// TwinCAT 3 PLC project AdsGo_Det
// ProgramVersion: 3.1.4026.21
// libraries:
//   Tc2_Standard, * (Beckhoff Automation GmbH)
//   Tc2_System, * (Beckhoff Automation GmbH)
//   Tc3_Module, * (Beckhoff Automation GmbH)
// project tree:
//   Lib/ TestStruct.TcDUT, PackNone.TcDUT, PackTwo.TcDUT, PackFour.TcDUT, PackEight.TcDUT, StructTests.TcPOU, Deterministic.TcPOU
//   Programs/ Main.TcPOU
//   Tasks/ PlcTask.TcTTO
// real-time tasks:
//   TASK PlcTask: cycle T#10ms, priority 20, ADS port 354

CONFIGURATION AdsGo_Det
    RESOURCE PLC ON TwinCAT3
        TASK PlcTask(INTERVAL := T#10ms, PRIORITY := 20);
        PROGRAM Main WITH PlcTask : Main;
    END_RESOURCE
END_CONFIGURATION

// ---- Lib/TestStruct.TcDUT
TYPE TestStruct :
STRUCT
	seed       : UDINT;
	bool_var   : BOOL;
	sint_var   : SINT;
	usint_var  : USINT;
	byte_var   : BYTE;
	int_var    : INT;
	uint_var   : UINT;
	word_var   : WORD;
	dint_var   : DINT;
	udint_var  : UDINT;
	dword_var  : DWORD;
	lint_var   : LINT;
	ulint_var  : ULINT;
	lword_var  : LWORD;
	real_var   : REAL;
	lreal_var  : LREAL;
	time_var   : TIME;
	tod_var    : TOD;
	date_var   : DATE;
	dt_var     : DT;
	//ltime_var : LTIME;
	//ltod_var  : LTOD;
	//ldate_var : LDATE;
	//ldt_var   : LDT;
	string_var : STRING(255);
END_STRUCT
END_TYPE

// ---- Lib/PackNone.TcDUT
{attribute 'pack_mode' := '0'}
TYPE PackNone :
STRUCT
	b1  : BOOL;
	d1  : DWORD;
	b2  : BOOL;
	lw1 : LWORD;
END_STRUCT
END_TYPE

// ---- Lib/PackTwo.TcDUT
{attribute 'pack_mode' := '2'}
TYPE PackTwo :
STRUCT
	b1  : BOOL;
	d1  : DWORD;
	b2  : BOOL;
	lw1 : LWORD;
END_STRUCT
END_TYPE

// ---- Lib/PackFour.TcDUT
{attribute 'pack_mode' := '4'}
TYPE PackFour :
STRUCT
	b1  : BOOL;
	d1  : DWORD;
	b2  : BOOL;
	lw1 : LWORD;
END_STRUCT
END_TYPE

// ---- Lib/PackEight.TcDUT
{attribute 'pack_mode' := '8'}
TYPE PackEight :
STRUCT
	b1  : BOOL;
	d1  : DWORD;
	b2  : BOOL;
	lw1 : LWORD;
END_STRUCT
END_TYPE

// ---- Programs/Main.TcPOU
PROGRAM Main
VAR
	test : Deterministic;

	// Writable targets — PLC never modifies these, Go test owns them
	write_bool_var   : BOOL;
	write_sint_var   : SINT;
	write_usint_var  : USINT;
	write_byte_var   : BYTE;
	write_int_var    : INT;
	write_uint_var   : UINT;
	write_word_var   : WORD;
	write_dint_var   : DINT;
	write_udint_var  : UDINT;
	write_dword_var  : DWORD;
	write_lint_var   : LINT;
	write_ulint_var  : ULINT;
	write_lword_var  : LWORD;
	write_real_var   : REAL;
	write_lreal_var  : LREAL;
	write_time_var   : TIME;
	write_tod_var    : TOD;
	write_date_var   : DATE;
	write_dt_var     : DT;
	//write_ltime_var  : LTIME;
	//write_ltod_var   : LTOD;
	//write_ldate_var  : LDATE;
	//write_ldt_var    : LDT;
	write_string_var : STRING(255);
	write_struct_var : TestStruct;
	write_int_array  : ARRAY[0..9] OF INT;
	write_dint_array : ARRAY[0..9] OF DINT;
	write_2d_array   : ARRAY[0..2, 0..2] OF INT;

	// Struct packing test targets — one instance per pack_mode
	// struct_tests: PLC drives these from seed (Go read-only for phase 1)
	struct_tests : StructTests;
	// pack_*: Go-owned write targets (PLC never modifies, used in phase 2)
	pack_none  : PackNone;
	pack_two   : PackTwo;
	pack_four  : PackFour;
	pack_eight : PackEight;
END_VAR

test();
struct_tests();

END_PROGRAM

// ---- Lib/Deterministic.TcPOU
FUNCTION_BLOCK Deterministic
VAR
	// Control (writable by Go test)
	seed               : UDINT := 0;
	auto_mode          : BOOL := FALSE;
	auto_tick_interval : UDINT := 50;

	// Outputs
	bool_var   : BOOL;
	sint_var   : SINT;
	usint_var  : USINT;
	byte_var   : BYTE;
	int_var    : INT;
	uint_var   : UINT;
	word_var   : WORD;
	dint_var   : DINT;
	udint_var  : UDINT;
	dword_var  : DWORD;
	lint_var   : LINT;
	ulint_var  : ULINT;
	lword_var  : LWORD;
	real_var   : REAL;
	lreal_var  : LREAL;
	time_var   : TIME;
	tod_var    : TOD;
	date_var   : DATE;
	dt_var     : DT;
	//ltime_var  : LTIME;
	//ltod_var   : LTOD;
	//ldate_var  : LDATE;
	//ldt_var    : LDT;
	string_var : STRING(255);
	struct_var : TestStruct;
	int_array  : ARRAY[0..9] OF INT;
	dint_array : ARRAY[0..9] OF DINT;
	array_2d   : ARRAY[0..2, 0..2] OF INT;

	// Private
	_tick_counter : UDINT;
	_i            : UDINT;
	_j            : UDINT;
END_VAR

// -----------------------------------------------------------------------
// Auto-increment mode: advance seed every auto_tick_interval cycles
// -----------------------------------------------------------------------
IF auto_mode THEN
	IF _tick_counter >= auto_tick_interval THEN
		seed          := seed + 1;
		_tick_counter := 0;
	ELSE
		_tick_counter := _tick_counter + 1;
	END_IF
END_IF

// -----------------------------------------------------------------------
// Update variables — all fields are deterministic functions of seed
// -----------------------------------------------------------------------
bool_var  := (seed MOD 2 = 0);
sint_var  := UDINT_TO_SINT(seed);
usint_var := UDINT_TO_USINT(seed);
byte_var  := UDINT_TO_BYTE(seed);
int_var   := UDINT_TO_INT(seed);
uint_var  := UDINT_TO_UINT(seed);
word_var  := UDINT_TO_WORD(seed);
dint_var  := UDINT_TO_DINT(seed);
udint_var := seed;
dword_var := UDINT_TO_DWORD(seed);
lint_var  := UDINT_TO_LINT(seed);
ulint_var := UDINT_TO_ULINT(seed);
lword_var := UDINT_TO_LWORD(seed);
real_var  := UDINT_TO_REAL(seed);
lreal_var := UDINT_TO_LREAL(seed);

// Date/time types — raw truncating casts, same bit pattern Go test will verify
time_var  := UDINT_TO_TIME(seed);
tod_var   := UDINT_TO_TOD(seed MOD 86400000);
date_var  := UDINT_TO_DATE(seed);
dt_var    := UDINT_TO_DT(seed);
//ltime_var := ULINT_TO_LTIME(UDINT_TO_ULINT(seed));
//ltod_var  := ULINT_TO_LTOD(UDINT_TO_ULINT(seed) MOD 86400000000000);
//ldate_var := ULINT_TO_LDATE(UDINT_TO_ULINT(seed));
//ldt_var   := ULINT_TO_LDT(UDINT_TO_ULINT(seed));

string_var := CONCAT('S=', UDINT_TO_STRING(seed));

// -----------------------------------------------------------------------
// Update test struct — all fields are deterministic functions of seed
// -----------------------------------------------------------------------
struct_var.seed      := seed;

struct_var.bool_var  := bool_var;
struct_var.sint_var  := sint_var;
struct_var.usint_var := usint_var;
struct_var.byte_var  := byte_var;
struct_var.int_var   := int_var;
struct_var.uint_var  := uint_var;
struct_var.word_var  := word_var;
struct_var.dint_var  := dint_var;
struct_var.udint_var := udint_var;
struct_var.dword_var := dword_var;
struct_var.lint_var  := lint_var;
struct_var.ulint_var := ulint_var;
struct_var.lword_var := lword_var;
struct_var.real_var  := real_var;
struct_var.lreal_var := lreal_var;
struct_var.time_var  := time_var;
struct_var.tod_var   := tod_var;
struct_var.date_var  := date_var;
struct_var.dt_var    := dt_var;
//struct_var.ltime_var := ltime_var;
//struct_var.ltod_var  := ltod_var;
//struct_var.ldate_var := ldate_var;
//struct_var.ldt_var   := ldt_var;
struct_var.string_var := string_var;

// -----------------------------------------------------------------------
// Update 1-D arrays: element[i] = UDINT_TO_x(seed + i)
// -----------------------------------------------------------------------
FOR _i := 0 TO 9 DO
	int_array[_i]  := UDINT_TO_INT(seed + _i);
	dint_array[_i] := UDINT_TO_DINT(seed + _i);
END_FOR

// -----------------------------------------------------------------------
// Update 2-D array: element[i,j] = UDINT_TO_INT(seed + i*3 + j)
// -----------------------------------------------------------------------
FOR _i := 0 TO 2 DO
	FOR _j := 0 TO 2 DO
		array_2d[_i, _j] := UDINT_TO_INT(seed + _i * 3 + _j);
	END_FOR
END_FOR

END_FUNCTION_BLOCK

// ---- Lib/StructTests.TcPOU
FUNCTION_BLOCK StructTests
VAR
	seed       : UDINT;
	pack_none  : PackNone;
	pack_two   : PackTwo;
	pack_four  : PackFour;
	pack_eight : PackEight;
END_VAR

// All four structs share the same fields and the same seed-driven formula.
// b1  = (seed MOD 2 = 0)
// d1  = seed
// b2  = (seed MOD 3 = 0)
// lw1 = LWORD(seed) * LWORD(3)
pack_none.b1  := (seed MOD 2 = 0);
pack_none.d1  := seed;
pack_none.b2  := (seed MOD 3 = 0);
pack_none.lw1 := UDINT_TO_LWORD(seed) * UDINT_TO_LWORD(3);

pack_two.b1  := pack_none.b1;
pack_two.d1  := pack_none.d1;
pack_two.b2  := pack_none.b2;
pack_two.lw1 := pack_none.lw1;

pack_four.b1  := pack_none.b1;
pack_four.d1  := pack_none.d1;
pack_four.b2  := pack_none.b2;
pack_four.lw1 := pack_none.lw1;

pack_eight.b1  := pack_none.b1;
pack_eight.d1  := pack_none.d1;
pack_eight.b2  := pack_none.b2;
pack_eight.lw1 := pack_none.lw1;

END_FUNCTION_BLOCK
